Staubli VAL3: onStop.pgx

public program onStop(string& x_sItem[])
begin
  if x_sItem=="kill"
    // empty the ram
    pt:libLoad("Disk://kernel/template/session/saveTraj/HOME")
  endIf
end
